// TIA Portal V16 export
// export: Created 2024-04-26T21:24:44.8947955Z, ExportSetting WithDefaults, DisplayName Totally Integrated Automation Portal, DisplayVersion V16, DisplayName TIA Portal Version Control Interface, DisplayVersion V16, DisplayName TIA Portal Openness, DisplayVersion V16, DisplayName STEP 7 Professional, DisplayVersion V16, DisplayName STEP 7 Safety, DisplayVersion V16, DisplayName WinCC Professional, DisplayVersion V16
VAR_GLOBAL   // PLC tag table "Default tag table"
   Axis_1_Pulse AT %Q5.0 : Bool;
   Axis_2_Pulse AT %Q5.1 : Bool;
   Axis_2_Direction AT %Q5.5 : Bool;
   Axis_1_Direction AT %Q5.4 : Bool;
   Axis_3_Direction AT %Q5.6 : Bool;
   Axis_3_Pulse AT %Q5.2 : Bool;
   POLE AT %I10.0 : Bool;
   START AT %I10.1 : Bool;
   Czujnik_osi AT %I10.4 : Bool;
   PP_os1 AT %I10.5 : Bool;
   PL_os1 AT %I10.6 : Bool;
   HOME_os1 AT %I10.7 : Bool;
   PP_os2 AT %I11.0 : Bool;
   PL_os2 AT %I11.1 : Bool;
   HOME_os2 AT %I11.2 : Bool;
   PP_os3 AT %I11.3 : Bool;
   PL_os3 AT %I11.4 : Bool;
   HOME_os3 AT %I11.5 : Bool;
   GRA_ON AT %M0.1 : Bool;
   Ruch_HOME_os1 AT %M0.2 : Bool;
   Ruch_HOME_os2 AT %M0.3 : Bool;
   Ruch_HOME_os3 AT %M0.4 : Bool;
   RESET_bledow AT %M0.5 : Bool;
   warunek_sek2 AT %M2.2 : Bool;
   warunek_sek3 AT %M1.2 : Bool;
   licznik_os1 AT %MW1 : Int;
   Przycisk_POLE_ON AT %M1.3 : Bool;
   warunek_sek1 AT %M1.4 : Bool;
   Meta AT %I10.2 : Bool;
   Nowa_Gra_reset AT %I10.3 : Bool;
   Pozycja_0_osi1 AT %M3.0 : Bool;
   Pozycja0_osi2 AT %M3.1 : Bool;
   Pozycja0_osi3 AT %M3.2 : Bool;
   RESET AT %M3.3 : Bool;
   Zalaczenie_osi AT %M3.4 : Bool;
   tag AT %M3.5 : Bool;
   tag1 AT %M3.6 : Bool;
   tag2 AT %M3.7 : Bool;
   tag3 AT %M4.0 : Bool;
   tag4 AT %M4.1 : Bool;
   tag5 AT %M4.2 : Bool;
   tag6 AT %M4.3 : Bool;
   LEWO AT %M4.4 : Bool;
   PRAWO AT %M4.5 : Bool;
   Tag_1 AT %I100.0 : Bool;
END_VAR
